Yaskawa INFORM job: _DEL24.JBI

/JOB
//NAME _DEL24
//POS
///NPOS 0,0,0,0,0,1
///TOOL 0
///POSTYPE ANGLE
///ANGLE
EX00110=0.0000
//INST
///DATE 2018/08/30 12:42
///ATTR SC,RW,SY
///GROUP1 ST2
///LVARS 5,0,5,0,0,0,0,0
NOP
*top
GETS PX111 $PX001
GETE LD000 EX110 (1)
DIV LD000 20000
SET LB000 LD000
DOUT OG#(83) LB000
DELAY 200
JUMP *top
END
